(* CODESYS project betu_rendezes

Project tree, tasks and I/O mapping:
  Device : CODESYS Control Win V3 x64, 3S - Smart Software Solutions GmbH, version 3.5.19.70
    application Application
      libraries: Standard, 3.5.18.0 (System)
      task MainTask (cyclic, interval t#20ms, priority 1) calls PLC_PRG, TRIGER
      function BETWEEN [ST]
      data type ENU_BETU
      data type ENUCONV2
      data type ENUCONV
      data type ENUFBCSERE
      data type ENUFBFELVESZ
      data type ENUFBLERAK
      data type ENUFELVESZ_LERAK
      data type ENUREAD
      data type ENUROBOT
      data type ENUSCAN
      function block FBCONV2 [ST]
      function block FBCONV [ST]
      function block FBCSERE [ST]
      function block FBFELVESZ [ST]
      function block FBFELVESZ_LERAK [ST]
      function block FBLERAK [ST]
      function block FBREAD [ST]
      function block FBROBOT [ST]
      function block FBSCAN [ST]
      global variables GVL
      global variables I
      program PLC_PRG [ST]
      global variables Q
      data type STATE
      data type SZALAG_ENU
      program TRIGER [ST]
      function block VILLOGO4 [ST]
    Ethernet : Ethernet, CODESYS, version 4.2.0.0
        settings: IPAddress = [127,0,0,1]; SubnetMask = [255,255,255,0]; GatewayAddress = [0,0,0,0]; MACAddress = [16#00,16#00,16#00,16#00,16#00,16#00]; SaveCommunicationSettings = FALSE; IPAddress = [192,168,0,2]; SubnetMask = [255,255,255,0]; GatewayAddress = [0,0,0,0]
      ModbusTCP_Slave_Device : ModbusTCP Slave Device, 3S - Smart Software Solutions GmbH, version 4.3.0.0
          settings: Coils Size = 20; Discrete Inputs Size = 20; StartAdresses.HoldingRegister = 20; StartAdresses.InputRegister = 20
          unmapped channels: %IW20 Holding Registers, %QW20 Input Registers
    Pfc200Bus : Wago PFC200 internal bus, 3S - Smart Software Solutions GmbH, version 4.1.0.0
      _750_14xx_1 : 16DI, WAGO Kontakttechnik GmbH u. Co. KG, order no. 750-14xx, version 4.1.0.0
          unmapped channels: %IW10 Digital Inputs 0 - 15
      _750_14xx : 16DI, WAGO Kontakttechnik GmbH u. Co. KG, order no. 750-14xx, version 4.1.0.0
          unmapped channels: %IW5 Digital Inputs 0 - 15
      _750_15xx_1 : 16DO, WAGO Kontakttechnik GmbH u. Co. KG, order no. 750-15xx, version 4.1.0.0
          unmapped channels: %QW10 Digital Outputs 0 - 15
      _750_15xx : 16DO, WAGO Kontakttechnik GmbH u. Co. KG, order no. 750-15xx, version 4.1.0.0
          unmapped channels: %QW5 Digital Outputs 0 - 15
      _75x_459 : 75x-459/0..-000 4AI, 0-10 V, WAGO Kontakttechnik GmbH u. Co. KG, order no. 75x-459(/0..-000), version 4.1.0.0
          unmapped channels: Analog Input Channel 0, Analog Input Channel 1, Analog Input Channel 2, Analog Input Channel 3
      _75x_559 : 75x-559/0..-000 4AO, 0-10 V, WAGO Kontakttechnik GmbH u. Co. KG, order no. 75x-559(/0..-000), version 4.1.0.0
          unmapped channels: Analog Output Channel 0, Analog Output Channel 1, Analog Output Channel 2, Analog Output Channel 3
    Pfc200Bus : Wago PFC200 internal bus, 3S - Smart Software Solutions GmbH, version 4.1.0.0
      _750_14xx_1 : 16DI, WAGO Kontakttechnik GmbH u. Co. KG, order no. 750-14xx, version 4.1.0.0
          unmapped channels: %IW20 Digital Inputs 0 - 15
      _750_14xx : 16DI, WAGO Kontakttechnik GmbH u. Co. KG, order no. 750-14xx, version 4.1.0.0
          unmapped channels: Digital Inputs 0 - 15
      _750_15xx : 16DO, WAGO Kontakttechnik GmbH u. Co. KG, order no. 750-15xx, version 4.1.0.0
          unmapped channels: Digital Outputs 0 - 15
      _750_15xx_1 : 16DO, WAGO Kontakttechnik GmbH u. Co. KG, order no. 750-15xx, version 4.1.0.0
          unmapped channels: %QW20 Digital Outputs 0 - 15
      _75x_459 : 75x-459/0..-000 4AI, 0-10 V, WAGO Kontakttechnik GmbH u. Co. KG, order no. 75x-459(/0..-000), version 4.1.0.0
          unmapped channels: Analog Input Channel 0, Analog Input Channel 1, Analog Input Channel 2, Analog Input Channel 3
      _75x_559 : 75x-559/0..-000 4AO, 0-10 V, WAGO Kontakttechnik GmbH u. Co. KG, order no. 75x-559(/0..-000), version 4.1.0.0
          unmapped channels: Analog Output Channel 0, Analog Output Channel 1, Analog Output Channel 2, Analog Output Channel 3
  Device : CODESYS Control for PFC200 SL, 3S - Smart Software Solutions GmbH, version 4.1.0.0
    application Application
      libraries: Standard, 3.5.18.0 (System)
      task MainTask (cyclic, interval t#20ms, priority 1) calls PLC_PRG
      program PLC_PRG [ST]
    Pfc200Bus : Wago PFC200 internal bus, 3S - Smart Software Solutions GmbH, version 4.1.0.0
*)

// Device/Application/ENU_BETU
{attribute 'qualified_only'}
//{attribute 'strict'}
TYPE ENU_BETU :
(
	A := 0,
	B := 1,
	C := 2, 
	D := 3,
	E := 4,
	F := 5,
	G := 6,
	H := 7,
	FASZ := 9999
);
END_TYPE

// Device/Application/ENUCONV2
{attribute 'qualified_only'}
//{attribute 'strict'}
TYPE ENUCONV2:
(
	PRESET := 0,
	MOZGAS1 := 1,
	MOZGAS2 := 2,
	DONE := 3,
	WAIT := 4
);
END_TYPE

// Device/Application/ENUCONV
{attribute 'qualified_only'}
//{attribute 'strict'}
TYPE ENUCONV:
(
	PRESET := 0,
	MOZGAS_START := 1,
	MOZGAS_DONE := 2
);
END_TYPE

// Device/Application/ENUFBCSERE
{attribute 'qualified_only'}
//{attribute 'strict'}
TYPE ENUFBCSERE:
(
	PRESET := 0,
	HONNA_TEMP1 := 1,
	HOVA_HONNA := 2,
	TEMP1_HOVA := 3,
	DONE := 4
);
END_TYPE

// Device/Application/ENUFBFELVESZ
{attribute 'qualified_only'}
//{attribute 'strict'}
TYPE ENUFBFELVESZ:
(
	PRESET := 0,
	DONTTES := 1,
	MOZO_1 := 2,
	FELVESZ := 3,
	VISSZA_MOZOG := 4,
	DONE := 5
);
END_TYPE

// Device/Application/ENUFBLERAK
{attribute 'qualified_only'}
//{attribute 'strict'}
TYPE ENUFBLERAK:
(
	PRESET := 0,
	DONTTES := 1,
	MOZO_1 := 2,
	LERAK := 3,
	VISSZA_MOZOG := 4,
	DONE := 5
);
END_TYPE

// Device/Application/ENUFELVESZ_LERAK
{attribute 'qualified_only'}
//{attribute 'strict'}
TYPE ENUFELVESZ_LERAK:
(
	PRESET := 0,
	MOZGAT_1 := 1,
	FELVESZ_1 := 2,
	LERAAK_1 := 3,
	MOZOG_2 := 4,
	MOZOG_3 := 5,
	DONTES := 6,
	WAIT := 7,
	DONE := 8
);
END_TYPE

// Device/Application/ENUREAD
{attribute 'qualified_only'}
//{attribute 'strict'}
TYPE ENUREAD:
(
	PRESET := 0,
	FELVESZ := 1,
	OLVASASHOZ_MEGY_WAIT := 2,
	LERAK := 3,
	SZALAG_VISSZA := 4,
	OLVASASHOZ_MEGY := 5,
	OLVAS := 6,
	LERAK_WAIT := 7,
	SZALAG_ODA := 8,
	DONE := 9
);
END_TYPE

// Device/Application/ENUROBOT
{attribute 'qualified_only'}
//{attribute 'strict'}
TYPE ENUROBOT:
(
	PRESET := 0,
	MOZGAS_START := 1,
	MOZGAS_DONE := 2
);
END_TYPE

// Device/Application/ENUSCAN
{attribute 'qualified_only'}
//{attribute 'strict'}
TYPE ENUSCAN:
(
	PRESET := 0,
	MOZGAS_START := 1,
	MOZGAS_DONE := 2
);
END_TYPE

// Device/Application/STATE
{attribute 'qualified_only'}
//{attribute 'strict'}
TYPE STATE:
(
	PRESET := 0,
	BEOLVAS := 1,
	CIKLUS := 2,
	CSERE := 3
);
END_TYPE

// Device/Application/SZALAG_ENU
{attribute 'qualified_only'}
{attribute 'strict'}
TYPE SZALAG_ENU :
(
	TEMP1 := 0,
	EGY := 1,
	KETO := 2,
	HAROM := 3, 
	NEGY := 4,
	OT := 5,
	HAT := 6,
	HET := 7,
	NYOLC := 8,
	TEMP2 := 9
);
END_TYPE

// Device/Application/GVL
{ attribute 'qualified_only'}
VAR_GLOBAL
   CHAR_0_R_TRIG : R_TRIG;
   CHAR_0_F_TRIG : F_TRIG;
   CHAR_1_R_TRIG : R_TRIG;
   CHAR_1_F_TRIG : F_TRIG;
   CHAR_2_R_TRIG : R_TRIG;
   CHAR_2_F_TRIG : F_TRIG;
   RFID_RUN_R_TRIG : R_TRIG;
   RFID_RUN_F_TRIG : F_TRIG;
   RFID_DONE_R_TRIG : R_TRIG;
   RFID_DONE_F_TRIG : F_TRIG;
   ROBOT_ACTUAL_0_R_TRIG : R_TRIG;
   ROBOT_ACTUAL_0_F_TRIG : F_TRIG;
   ROBOT_ACTUAL_1_R_TRIG : R_TRIG;
   ROBOT_ACTUAL_1_F_TRIG : F_TRIG;
   ROBOT_ACTUAL_2_R_TRIG : R_TRIG;
   ROBOT_ACTUAL_2_F_TRIG : F_TRIG;
   ROBOT_RUN_R_TRIG : R_TRIG;
   ROBOT_RUN_F_TRIG : F_TRIG;
   ROBOT_DONE_R_TRIG : R_TRIG;
   ROBOT_DONE_F_TRIG : F_TRIG;
   CONV_RUN_R_TRIG : R_TRIG;
   CONV_DONE_R_TRIG : R_TRIG;
   CONV_DONE_F_TRIG : F_TRIG;
   START_R_TRIG : R_TRIG;
   START_F_TRIG : F_TRIG;
   STOP_R_TRIG : R_TRIG;
   STOP_F_TRIG : F_TRIG;
   
   
   SZALAG : ARRAY[0..9] OF ENU_BETU := [10(ENU_BETU.FASZ)] ;
   SZALAG_OFFSET : INT;
   
   STATE : STATE;
   
END_VAR

// Device/Application/I
{attribute 'qualified_only'}
VAR_GLOBAL
END_VAR

// Device/Application/Q
{attribute 'qualified_only'}
VAR_GLOBAL
END_VAR

// Device/Application/PLC_PRG
PROGRAM PLC_PRG
VAR
	
END_VAR

END_PROGRAM

// Device/Application/PLC_PRG
PROGRAM PLC_PRG
VAR
END_VAR

END_PROGRAM

// Device/Application/TRIGER
PROGRAM TRIGER
VAR
END_VAR

GVL.CHAR_0_R_TRIG(CLK:= I.CHAR_0);
GVL.CHAR_0_F_TRIG(CLK:= I.CHAR_0);
GVL.CHAR_1_R_TRIG(CLK:= I.CHAR_1);
GVL.CHAR_1_F_TRIG(CLK:= I.CHAR_1);
GVL.CHAR_2_R_TRIG(CLK:= I.CHAR_2);
GVL.CHAR_2_F_TRIG(CLK:= I.CHAR_2);
GVL.RFID_RUN_R_TRIG(CLK:= I.RFID_RUN);
GVL.RFID_RUN_F_TRIG(CLK:= I.RFID_RUN);
GVL.RFID_DONE_R_TRIG(CLK:= I.RFID_DONE);
GVL.RFID_DONE_F_TRIG(CLK:= I.RFID_DONE);
GVL.ROBOT_ACTUAL_0_R_TRIG(CLK:= I.ROBOT_ACTUAL_0);
GVL.ROBOT_ACTUAL_0_F_TRIG(CLK:= I.ROBOT_ACTUAL_0);
GVL.ROBOT_ACTUAL_1_R_TRIG(CLK:= I.ROBOT_ACTUAL_1);
GVL.ROBOT_ACTUAL_1_F_TRIG(CLK:= I.ROBOT_ACTUAL_1);
GVL.ROBOT_ACTUAL_2_R_TRIG(CLK:= I.ROBOT_ACTUAL_2);
GVL.ROBOT_ACTUAL_2_F_TRIG(CLK:= I.ROBOT_ACTUAL_2);
GVL.ROBOT_RUN_R_TRIG(CLK:= I.ROBOT_RUN);
GVL.ROBOT_RUN_F_TRIG(CLK:= I.ROBOT_RUN);
GVL.ROBOT_DONE_R_TRIG(CLK:= I.ROBOT_DONE);
GVL.ROBOT_DONE_F_TRIG(CLK:= I.ROBOT_DONE);
GVL.CONV_RUN_R_TRIG(CLK:= I.CONV_RUN);
GVL.CONV_DONE_R_TRIG(CLK:= I.CONV_DONE);
GVL.CONV_DONE_F_TRIG(CLK:= I.CONV_DONE);
GVL.START_R_TRIG(CLK:= I.START);
GVL.START_F_TRIG(CLK:= I.START);
GVL.STOP_R_TRIG(CLK:= I.STOP);
GVL.STOP_F_TRIG(CLK:= I.STOP);

END_PROGRAM

// Device/Application/BETWEEN
FUNCTION BETWEEN : BOOL
VAR_INPUT
	STATE : INT;
	LOW : INT;
	HIGH : INT;
END_VAR
VAR_OUTPUT
END_VAR
VAR
	EN_TRIG : F_TRIG;
END_VAR

IF STATE >= LOW AND STATE <= HIGH THEN
	BETWEEN := TRUE;
ELSE 
	BETWEEN := FALSE;
END_IF

END_FUNCTION

// Device/Application/FBCONV2
FUNCTION_BLOCK FBCONV2
VAR_INPUT
	EN : BOOL;
	IRANY : BOOL;
END_VAR
VAR_OUTPUT
	DONE  : BOOL;
END_VAR
VAR
	CONV2 : ENUCONV2;
	MOZGAT : FBCONV;
END_VAR

IF NOT EN THEN
	CONV2 := ENUCONV2.PRESET;
	RETURN;
END_IF

MOZGAT(IRANY := IRANY, EN:= (CONV2 = ENUCONV2.MOZGAS1) OR (CONV2 = ENUCONV2.MOZGAS2));

CASE CONV2 OF

	ENUCONV2.PRESET:
	IF TRUE THEN
		CONV2 := ENUCONV2.MOZGAS1;
	END_IF


	ENUCONV2.MOZGAS1:
	IF MOZGAT.DONE THEN
		CONV2 := ENUCONV2.WAIT;
	END_IF


	ENUCONV2.MOZGAS2:
	IF MOZGAT.DONE THEN
		CONV2 := ENUCONV2.DONE;
	END_IF
	

	ENUCONV2.WAIT:
	IF NOT MOZGAT.DONE THEN
		CONV2 := ENUCONV2.MOZGAS2;
	END_IF

END_CASE

DONE := (CONV2 = ENUCONV2.DONE);

END_FUNCTION_BLOCK

// Device/Application/FBCONV
FUNCTION_BLOCK FBCONV
VAR_INPUT
	EN : BOOL;
	IRANY : BOOL;
END_VAR
VAR_OUTPUT
	DONE  : BOOL;
END_VAR
VAR
	CONV : ENUCONV;
	TRANS_PRESET_MOZGAS_START_T : TON;
END_VAR

TRANS_PRESET_MOZGAS_START_T(PT:= T#100MS, IN:= (CONV = ENUCONV.PRESET));
IF NOT EN THEN
	CONV := ENUCONV.PRESET;
	DONE := FALSE;
	RETURN;
END_IF



CASE CONV OF

	ENUCONV.PRESET:
	IF IRANY THEN
		Q.CONV_RIGHT := TRUE;
		Q.CONV_LEFT := FALSE;
	ELSE
		Q.CONV_RIGHT := FALSE;
		Q.CONV_LEFT := TRUE;
	END_IF

	IF TRANS_PRESET_MOZGAS_START_T.Q THEN
		CONV := ENUCONV.MOZGAS_START;
	END_IF

	ENUCONV.MOZGAS_START:

	IF gvl.CONV_DONE_R_TRIG.Q AND NOT I.CONV_RUN THEN
		CONV := ENUCONV.MOZGAS_DONE;
	END_IF

	ENUCONV.MOZGAS_DONE:


END_CASE

DONE := (CONV = ENUCONV.MOZGAS_DONE);
Q.CONV_START := (CONV = ENUCONV.MOZGAS_START);

END_FUNCTION_BLOCK

// Device/Application/FBCSERE
FUNCTION_BLOCK FBCSERE
VAR_INPUT
	EN : BOOL;
	HONNAN : INT;
	HOVA : INT;
END_VAR
VAR_OUTPUT
	DONE:BOOL;
END_VAR
VAR
	FBCSERE : ENUFBCSERE;
	FELLE1 : FBFELVESZ_LERAK;
	FELLE2 : FBFELVESZ_LERAK;
	FELLE3 : FBFELVESZ_LERAK;
END_VAR

FELLE1(EN:= (FBCSERE = ENUFBCSERE.HONNA_TEMP1) , HONNAN := HONNAN , HOVA := SZALAG_ENU.TEMP1);
FELLE2(EN:= (FBCSERE = ENUFBCSERE.HOVA_HONNA) , HONNAN := HOVA , HOVA := HONNAN);
FELLE3(EN:= (FBCSERE = ENUFBCSERE.TEMP1_HOVA) , HONNAN := SZALAG_ENU.TEMP1 , HOVA := HOVA );
DONE := (FBCSERE = ENUFBCSERE.DONE);
IF NOT EN THEN
	FBCSERE := ENUFBCSERE.PRESET;
	DONE := FALSE;
	RETURN;
END_IF



CASE FBCSERE OF

	ENUFBCSERE.PRESET:
	IF EN THEN
		FBCSERE := ENUFBCSERE.HONNA_TEMP1;
	END_IF


	ENUFBCSERE.HONNA_TEMP1:
	IF FELLE1.DONE THEN
		FBCSERE := ENUFBCSERE.HOVA_HONNA;
	END_IF


	ENUFBCSERE.HOVA_HONNA:
	IF FELLE2.DONE THEN
		FBCSERE := ENUFBCSERE.TEMP1_HOVA;
	END_IF


	ENUFBCSERE.TEMP1_HOVA:
	IF FELLE3.DONE THEN
		FBCSERE := ENUFBCSERE.DONE;
	END_IF


	ENUFBCSERE.DONE:
END_CASE

END_FUNCTION_BLOCK

// Device/Application/FBFELVESZ_LERAK
FUNCTION_BLOCK FBFELVESZ_LERAK
VAR_INPUT
	EN : BOOL;
	HONNAN : SZALAG_ENU ;
	HOVA : SZALAG_ENU ;
END_VAR
VAR_OUTPUT
	DONE : BOOL;
END_VAR
VAR

	FBFELVESZ_LERAK : ENUFELVESZ_LERAK;
	FELVESZ_LERAK : FBROBOT;
	J : INT;
	K : INT;
	MOZGAS_1_CONV : FBCONV2;
	MOZGAS_1_KEL : BOOL;
	MOZOG_2_KELL : BOOL;
	TRANS_WAIT_LERAAK_1_T : TON;
	FELVESZ_HELY : INT;
	OFFSET : INT;
	IRANY : BOOL;
	ROBOT_TARGET :INT;
END_VAR

IF NOT EN THEN
	FBFELVESZ_LERAK := ENUFELVESZ_LERAK.PRESET;
	DONE := FALSE;
	OFFSET := 0;
	MOZGAS_1_KEL := FALSE;
	MOZOG_2_KELL := FALSE;
	RETURN;
	
END_IF

TRANS_WAIT_LERAAK_1_T(PT:= T#200MS, IN:= (FBFELVESZ_LERAK = ENUFELVESZ_LERAK.WAIT));
MOZGAS_1_CONV(EN:= (FBFELVESZ_LERAK = ENUFELVESZ_LERAK.MOZGAT_1) OR (FBFELVESZ_LERAK = ENUFELVESZ_LERAK.MOZOG_2) OR (FBFELVESZ_LERAK = ENUFELVESZ_LERAK.MOZOG_3) , IRANY := IRANY ,DUPLA := ((OFFSET < -1) OR (OFFSET > 1)));
FELVESZ_LERAK(EN:= (FBFELVESZ_LERAK = ENUFELVESZ_LERAK.FELVESZ_1) OR (FBFELVESZ_LERAK = ENUFELVESZ_LERAK.LERAAK_1),TARGET := ROBOT_TARGET);

CASE FBFELVESZ_LERAK OF

	ENUFELVESZ_LERAK.PRESET:
	IF EN THEN
		FBFELVESZ_LERAK := ENUFELVESZ_LERAK.DONTES;
	END_IF

	ENUFELVESZ_LERAK.DONTES:
	
	CASE HONNAN OF
		SZALAG_ENU.TEMP1:
		
		IRANY := TRUE;
		OFFSET := +1;
		MOZGAS_1_KEL := TRUE;
		
		SZALAG_ENU.D:
		
		IRANY := FALSE;
		OFFSET := -1;
		MOZGAS_1_KEL := TRUE;
		
		SZALAG_ENU.E:
		
		IRANY := TRUE;
		OFFSET := +1;
		MOZGAS_1_KEL := TRUE;
		
		SZALAG_ENU.TEMP2:
		IRANY := FALSE;
		OFFSET := -1;
		MOZGAS_1_KEL := TRUE;
	
	END_CASE

	IF MOZGAS_1_KEL  THEN
		FBFELVESZ_LERAK := ENUFELVESZ_LERAK.MOZGAT_1;
	ELSIF NOT MOZGAS_1_KEL THEN
		FELVESZ_HELY := HONNAN;
		Q.ROBOT_PICKUP := TRUE;
		FBFELVESZ_LERAK := ENUFELVESZ_LERAK.FELVESZ_1;
	END_IF

	ENUFELVESZ_LERAK.MOZGAT_1:
	
	IF MOZGAS_1_CONV.DONE THEN
		ROBOT_TARGET := HONNAN + OFFSET;
		Q.ROBOT_PICKUP := TRUE;
		FBFELVESZ_LERAK := ENUFELVESZ_LERAK.FELVESZ_1;
	END_IF

	ENUFELVESZ_LERAK.FELVESZ_1:
	//CASE SZERKEZET IFFEKEL HOVA MOZGATJA LERAKÁS ELÖT
	//HONNAN VESZEK FEL FELVESZ_HELY
	CASE HOVA OF
		SZALAG_ENU.TEMP1:
		
		IRANY := TRUE;
		OFFSET := +1-OFFSET;
		MOZOG_2_KELL := TRUE;
		
		SZALAG_ENU.D:
		
		IRANY := FALSE;
		OFFSET := -1-OFFSET;
		MOZOG_2_KELL := TRUE;
		
		SZALAG_ENU.E:
		
		IRANY := TRUE;
		OFFSET := +1-OFFSET;
		MOZOG_2_KELL := TRUE;
		
		SZALAG_ENU.TEMP2:
		IRANY := FALSE;
		OFFSET := -1-OFFSET;
		MOZOG_2_KELL := TRUE;
	
	END_CASE

	IF FELVESZ_LERAK.DONE AND MOZOG_2_KELL THEN
		Q.ROBOT_PICKUP := FALSE;
		FBFELVESZ_LERAK := ENUFELVESZ_LERAK.MOZOG_2;
	ELSIF FELVESZ_LERAK.DONE AND NOT MOZOG_2_KELL THEN
		Q.ROBOT_PICKUP := FALSE;
		Q.ROBOT_DROP := TRUE;
		ROBOT_TARGET := HOVA + OFFSET;
		FBFELVESZ_LERAK := ENUFELVESZ_LERAK.WAIT;
	END_IF

	ENUFELVESZ_LERAK.LERAAK_1:
	//LERAKASI POZICIO IRASA

	IF FELVESZ_LERAK.DONE AND NOT (OFFSET = 0) THEN
		Q.ROBOT_DROP := FALSE;
		
		IF OFFSET < 0 THEN 
			IRANY := TRUE;
		ELSIF OFFSET > 0 THEN
			IRANY := FALSE;
		END_IF
		
		FBFELVESZ_LERAK := ENUFELVESZ_LERAK.MOZOG_3;
	ELSIF FELVESZ_LERAK.DONE AND (OFFSET = 0) THEN
		Q.ROBOT_DROP := FALSE;
		FBFELVESZ_LERAK := ENUFELVESZ_LERAK.DONE;
	END_IF


	ENUFELVESZ_LERAK.MOZOG_2:
	IF MOZGAS_1_CONV.DONE THEN
		FBFELVESZ_LERAK := ENUFELVESZ_LERAK.LERAAK_1;
	END_IF


	ENUFELVESZ_LERAK.MOZOG_3:
	IF MOZGAS_1_CONV.DONE THEN
		FBFELVESZ_LERAK := ENUFELVESZ_LERAK.DONE;
	END_IF

	ENUFELVESZ_LERAK.WAIT:
	IF TRANS_WAIT_LERAAK_1_T.Q THEN
		Q.ROBOT_DROP := TRUE;
		ROBOT_TARGET := HOVA + OFFSET;
		FBFELVESZ_LERAK := ENUFELVESZ_LERAK.LERAAK_1;
	END_IF


	ENUFELVESZ_LERAK.DONE:
	
END_CASE

END_FUNCTION_BLOCK

// Device/Application/FBROBOT
FUNCTION_BLOCK FBROBOT
VAR_INPUT
	EN : BOOL;
	TARGET : INT;
END_VAR
VAR_OUTPUT
	DONE  : BOOL;
END_VAR
VAR
	CONV : ENUCONV;
	ROBOT : ENUROBOT;
	TRANS_PRESET_MOZGAS_START_T : TON;
END_VAR

IF NOT EN THEN
	ROBOT := ENUROBOT.PRESET;
	RETURN;
END_IF

TRANS_PRESET_MOZGAS_START_T(PT:= T#100MS, IN:= (ROBOT = ENUROBOT.PRESET));

CASE ROBOT OF

	ENUROBOT.PRESET:
	Q.ROBOT_POZ_2 := TARGET.2;
	Q.ROBOT_POZ_1 := TARGET.1;
	Q.ROBOT_POZ_0 := TARGET.0;

	IF TRANS_PRESET_MOZGAS_START_T.Q THEN
		ROBOT := ENUROBOT.MOZGAS_START;
	END_IF

	ENUROBOT.MOZGAS_START:
	Q.ROBOT_MOVE_START := TRUE;

	IF I.ROBOT_DONE AND NOT I.ROBOT_RUN THEN
		ROBOT := ENUROBOT.MOZGAS_DONE;
	END_IF

	ENUROBOT.MOZGAS_DONE:
	Q.ROBOT_MOVE_START := FALSE;

END_CASE

DONE := (ROBOT = ENUROBOT.MOZGAS_DONE);

END_FUNCTION_BLOCK

// Device/Application/FBFELVESZ
FUNCTION_BLOCK FBFELVESZ
VAR_INPUT
	EN : BOOL;
	HONNAN : INT;;
END_VAR
VAR_OUTPUT
		DONE  : BOOL;
		BETU :INT;
END_VAR
VAR

	FBFELVESZ : ENUFBFELVESZ;
	FELVESZ : FBROBOT;
	MOZGAS : FBCONV2;
	MOZGAS_KEL : BOOL;
	IRANY : BOOL;
	OFFSET : INT ;
END_VAR

MOZGAS(EN:= (FBFELVESZ = ENUFBFELVESZ.MOZO_1) OR (FBFELVESZ = ENUFBFELVESZ.VISSZA_MOZOG) , IRANY := IRANY ,DUPLA := FALSE);
FELVESZ(EN:= (FBFELVESZ = ENUFBFELVESZ.FELVESZ) , TARGET := HONNAN + OFFSET);
DONE := (FBFELVESZ = ENUFBFELVESZ.DONE);

IF NOT EN THEN
	FBFELVESZ := ENUFBFELVESZ.PRESET;
	DONE := FALSE ;
	OFFSET := 0;
	RETURN;
END_IF



CASE FBFELVESZ OF

	ENUFBFELVESZ.PRESET:
	IF EN THEN
		FBFELVESZ := ENUFBFELVESZ.DONTTES;
	END_IF


	ENUFBFELVESZ.DONTTES:
	
	CASE HONNAN OF
			SZALAG_ENU.TEMP1:
			
			IRANY := TRUE;
			OFFSET := 1;
			MOZGAS_KEL := TRUE;
			
			SZALAG_ENU.D:
			
			IRANY := FALSE;
			OFFSET := -1;
			MOZGAS_KEL := TRUE;
			
			SZALAG_ENU.E:
			
			IRANY := TRUE;
			OFFSET := -2;
			MOZGAS_KEL := TRUE;
			
			SZALAG_ENU.TEMP2:
			IRANY := FALSE;
			OFFSET := -2;
			MOZGAS_KEL := TRUE;
			
			SZALAG_ENU.F:
			
			OFFSET := -2;
			SZALAG_ENU.G:
			
			OFFSET := -2;
			
			SZALAG_ENU.H:
			
			OFFSET := -2;
		
		END_CASE

	IF MOZGAS_KEL THEN
		FBFELVESZ := ENUFBFELVESZ.MOZO_1;
	ELSIF NOT MOZGAS_KEL THEN
		Q.ROBOT_PICKUP := TRUE;
		FBFELVESZ := ENUFBFELVESZ.FELVESZ;
	END_IF


	ENUFBFELVESZ.MOZO_1:
	IF MOZGAS.DONE THEN
		Q.ROBOT_PICKUP := TRUE;
		FBFELVESZ := ENUFBFELVESZ.FELVESZ;
	END_IF


	ENUFBFELVESZ.FELVESZ:
	BETU := GVL.SZALAG[HONNAN];
	
	
	IF FELVESZ.DONE AND MOZGAS_KEL THEN
		GVL.SZALAG[HONNAN] := ENU_BETU.FASZ;
		IRANY := NOT IRANY;
		Q.ROBOT_PICKUP := FALSE;
		FBFELVESZ := ENUFBFELVESZ.VISSZA_MOZOG;
	ELSIF FELVESZ.DONE AND NOT MOZGAS_KEL THEN
		GVL.SZALAG[HONNAN] := ENU_BETU.FASZ;
		Q.ROBOT_PICKUP := FALSE;
		FBFELVESZ := ENUFBFELVESZ.DONE;
	END_IF


	ENUFBFELVESZ.VISSZA_MOZOG:
	IF MOZGAS.DONE THEN
		FBFELVESZ := ENUFBFELVESZ.DONE;
	END_IF


	ENUFBFELVESZ.DONE:
END_CASE

END_FUNCTION_BLOCK

// Device/Application/FBLERAK
FUNCTION_BLOCK FBLERAK
VAR_INPUT
		EN : BOOL;
		HOVA : INT;
		BETU : INT;
END_VAR
VAR_OUTPUT
END_VAR
VAR
	DONE  : BOOL;
	FBFELVESZ : ENUFBFELVESZ;
	FBLERAK : ENUFBLERAK;
	FELVESZ : FBROBOT;
	LERAK : FBROBOT;
	MOZGAS : FBCONV2;
	MOZGAS_KEL : BOOL;
	OFFSET : INT;
	IRANY : BOOL;
END_VAR

MOZGAS(EN:= (FBLERAK = ENUFBFELVESZ.MOZO_1) OR (FBLERAK = ENUFBFELVESZ.VISSZA_MOZOG) , IRANY := IRANY ,DUPLA := FALSE);
LERAK(EN:= (FBLERAK = ENUFBLERAK.LERAK),TARGET :=  (HOVA +OFFSET) );
IF NOT EN THEN
	FBLERAK := ENUFBLERAK.PRESET;
	DONE := FALSE;
	OFFSET := 0;
	
	RETURN;
END_IF



CASE FBLERAK OF

	ENUFBLERAK.PRESET:
	IF EN THEN
		FBLERAK := ENUFBLERAK.DONTTES;
	END_IF


	ENUFBLERAK.DONTTES:
	CASE HOVA OF
	SZALAG_ENU.TEMP1:
			
			IRANY := TRUE;
			OFFSET := 1;
			MOZGAS_KEL := TRUE;
			
			SZALAG_ENU.D:
			
			IRANY := FALSE;
			OFFSET := -1;
			MOZGAS_KEL := TRUE;
			
			SZALAG_ENU.E:
			
			IRANY := TRUE;
			OFFSET := -2;
			MOZGAS_KEL := TRUE;
			
			SZALAG_ENU.TEMP2:
			IRANY := FALSE;
			OFFSET := -3;
			MOZGAS_KEL := TRUE;
			
			SZALAG_ENU.F:
			
			OFFSET := -2;
			SZALAG_ENU.G:
			
			OFFSET := -2;
			
			SZALAG_ENU.H:
			
			OFFSET := -2;
		
		END_CASE

	IF MOZGAS_KEL THEN
		Q.ROBOT_DROP:= TRUE;
		FBLERAK := ENUFBLERAK.MOZO_1;
	ELSIF NOT MOZGAS_KEL THEN
		Q.ROBOT_DROP:= TRUE;
		FBLERAK := ENUFBLERAK.LERAK;
	END_IF


	ENUFBLERAK.MOZO_1:
	IF MOZGAS.DONE THEN
		FBLERAK := ENUFBLERAK.LERAK;
	END_IF


	ENUFBLERAK.LERAK:
	 GVL.SZALAG[HOVA] := BETU;
	IF LERAK.DONE AND MOZGAS_KEL THEN
		Q.ROBOT_DROP:= FALSE;
		IRANY := NOT IRANY;

		FBLERAK := ENUFBLERAK.VISSZA_MOZOG;
	ELSIF LERAK.DONE AND NOT MOZGAS_KEL THEN
		Q.ROBOT_DROP:= FALSE;
		FBLERAK := ENUFBLERAK.DONE;
	END_IF


	ENUFBLERAK.VISSZA_MOZOG:
	IF MOZGAS.DONE THEN
		FBLERAK := ENUFBLERAK.DONE;
	END_IF


	ENUFBLERAK.DONE:
END_CASE

DONE := (FBLERAK = ENUFBLERAK.DONE);

END_FUNCTION_BLOCK

// Device/Application/FBREAD
FUNCTION_BLOCK FBREAD
VAR_INPUT
	EN : BOOL;
END_VAR
VAR_OUTPUT
	DONE  : BOOL;
END_VAR
VAR
	CONV2 : FBCONV2;
	READ : ENUREAD;
	ROBOT : FBROBOT;
	ROBOT_POZ : INT;
	SCAN : FBSCAN;
	KOR : INT;
	TARGET_POZ : INT;
	IRANY : BOOL;
END_VAR

IF NOT EN THEN
	READ := ENUREAD.PRESET;
	DONE := FALSE;
	RETURN;
END_IF

CONV2(IRANY := IRANY, EN:= (READ = ENUREAD.SZALAG_ODA) OR (READ = ENUREAD.SZALAG_VISSZA));
ROBOT(TARGET := TARGET_POZ, EN:= (READ = ENUREAD.OLVASASHOZ_MEGY) OR (READ = ENUREAD.FELVESZ) OR (READ = ENUREAD.LERAK));
SCAN(BETU := (ROBOT_POZ MOD 7 - 1 + KOR), EN:= (READ = ENUREAD.OLVAS));

CASE READ OF
	ENUREAD.PRESET:
	Q.ROBOT_DROP := FALSE;
	Q.ROBOT_PICKUP := TRUE;
	ROBOT_POZ := 1;
	TARGET_POZ := ROBOT_POZ;

	IF TRUE THEN
		READ := ENUREAD.FELVESZ;
	END_IF


	ENUREAD.FELVESZ:
	IF ROBOT.DONE THEN
		Q.ROBOT_PICKUP := FALSE;

		READ := ENUREAD.OLVASASHOZ_MEGY_WAIT;
	END_IF


	ENUREAD.OLVASASHOZ_MEGY_WAIT:
	IF NOT ROBOT.DONE THEN
		TARGET_POZ := 7;
		READ := ENUREAD.OLVASASHOZ_MEGY;
	END_IF


	ENUREAD.LERAK:
	IF ROBOT.DONE THEN
		Q.ROBOT_PICKUP := TRUE;
		ROBOT_POZ := ROBOT_POZ + 1;

		READ := ENUREAD.LERAK_WAIT;
	END_IF


	ENUREAD.SZALAG_VISSZA:
	IF CONV2.DONE THEN
		READ := ENUREAD.DONE;
	END_IF


	ENUREAD.OLVASASHOZ_MEGY:
	IF ROBOT.DONE THEN
		IF ROBOT_POZ > 3 THEN
			KOR := 2;
		END_IF

		READ := ENUREAD.OLVAS;
	END_IF


	ENUREAD.OLVAS:
	IF SCAN.DONE THEN
		TARGET_POZ := ROBOT_POZ MOD 7;
		Q.ROBOT_DROP := TRUE;

		READ := ENUREAD.LERAK;
	END_IF


	ENUREAD.LERAK_WAIT:
	IF NOT (ROBOT_POZ = 11) AND NOT (ROBOT_POZ = 7) AND NOT ROBOT.DONE THEN
		READ := ENUREAD.FELVESZ;
	ELSIF ROBOT_POZ = 7 AND NOT ROBOT.DONE THEN
		ROBOT_POZ := 9;
		READ := ENUREAD.SZALAG_ODA;
	ELSIF ROBOT_POZ = 11 AND NOT ROBOT.DONE THEN
		READ := ENUREAD.SZALAG_VISSZA;
	END_IF
	TARGET_POZ := ROBOT_POZ;


	ENUREAD.SZALAG_ODA:
	IF CONV2.DONE THEN
		READ := ENUREAD.FELVESZ;
	END_IF

	ENUREAD.DONE:
	Q.ROBOT_PICKUP := FALSE;

END_CASE

DONE := (READ = ENUREAD.DONE);

END_FUNCTION_BLOCK

// Device/Application/FBSCAN
FUNCTION_BLOCK FBSCAN
VAR_INPUT
	EN : BOOL;
	BETU : INT;
END_VAR
VAR_OUTPUT
	DONE : BOOL;
END_VAR
VAR
	CONV : ENUCONV;
	ROBOT : ENUROBOT;
	SCAN : ENUSCAN;
	TRANS_PRESET_MOZGAS_START_T : TON;
END_VAR

IF NOT EN THEN
	SCAN := ENUSCAN.PRESET;
	DONE := FALSE;
	RETURN;
END_IF


CASE SCAN OF

	ENUSCAN.PRESET:
	IF TRUE THEN
		SCAN := ENUSCAN.MOZGAS_START;
	END_IF

	ENUSCAN.MOZGAS_START:
	GVL.SZALAG[BETU].0 := I.CHAR_0;
	GVL.SZALAG[BETU].1 := I.CHAR_1;
	GVL.SZALAG[BETU].2 := I.CHAR_2;
	Q.RFID_READ_START := TRUE;

	IF I.RFID_DONE AND NOT I.RFID_RUN THEN
		Q.RFID_READ_START := FALSE;;
		SCAN := ENUSCAN.MOZGAS_DONE;
	END_IF

	ENUSCAN.MOZGAS_DONE:

END_CASE

DONE := (SCAN = ENUSCAN.MOZGAS_DONE);

END_FUNCTION_BLOCK

// Device/Application/VILLOGO4
FUNCTION_BLOCK VILLOGO4
VAR_INPUT
	T1: TIME;
	T2: TIME;
	T3: TIME;
	T4: TIME;
END_VAR
VAR_IN_OUT
	Q1: BOOL;
	Q2: BOOL;
	Q3: BOOL;
	Q4: BOOL;
END_VAR
VAR
	T1_TON: TON;
	T2_TON: TON;
	T3_TON: TON;
	T4_TON: TON;
END_VAR
VAR_INPUT
	EN: BOOL := FALSE;
END_VAR
VAR
	EN_F_TRIG: F_TRIG;
	EN_R_TRIG: R_TRIG;
	STATE: INT := 0;
	PREV_STATE: INT := 0;
END_VAR

EN_F_TRIG(CLK := EN);
EN_R_TRIG(CLK := EN);

IF EN_F_TRIG.Q THEN
	Q1 := FALSE;
	Q2 := FALSE;
	Q3 := FALSE;
	Q4 := FALSE;
	T1_TON.PT := T1_TON.ET;
	T2_TON.PT := T2_TON.ET;
	T3_TON.PT := T3_TON.ET;
	T4_TON.PT := T4_TON.ET;
	STATE := 0;
ELSIF EN_R_TRIG.Q THEN
		Q1 := TRUE;
END_IF

IF NOT EN THEN
	RETURN;
END_IF

T1_TON(IN:= EN_R_TRIG.Q OR (STATE = 0), PT:= T1);
T2_TON(IN:= STATE = 1, PT:= T2);
T3_TON(IN:= STATE = 2, PT:= T3);
T4_TON(IN:= STATE = 3, PT:= T4);

IF T1_TON.Q THEN
	Q1 := FALSE;
	Q2 := TRUE;
END_IF
IF T2_TON.Q THEN
	Q2 := FALSE;
	Q3 := TRUE;
END_IF
IF T3_TON.Q THEN
	Q3 := FALSE;
	Q4 := TRUE;
END_IF
IF T4_TON.Q THEN
	Q4 := FALSE;
	Q1 := TRUE;
END_IF

IF T1_TON.Q OR T2_TON.Q OR T3_TON.Q OR T4_TON.Q THEN
	STATE := STATE + 1;
END_IF

IF STATE > 3 THEN
	STATE := 0;
END_IF

END_FUNCTION_BLOCK
